FUNCTION_BLOCK FB_InterlockManager

VAR
	aInterlocks: ARRAY[1..50] OF ST_Interlock;
	nIterator: INT := 1;
END_VAR

METHOD execute : BOOL
VAR_INPUT
END_VAR

VAR
	iterator: INT;

	
	Active:			BOOL;
	Bridge:			BOOL;
	SubjectDevice:	POINTER TO FB_BaseDevice;
	SubjectState:	E_DeviceState;
	Signal:			BOOL;
	Description: 	STRING(255);
	HoldSeq:		BOOL;
	InterlockType:	E_InterlockType;
	
	
	
END_VAR

FOR iterator:=1 TO nIterator BY 1 DO
	
	// Update local variable on each loop iteration
	
	Active := aInterlocks[iterator].Active;
	Bridge := aInterlocks[iterator].Bridge;
	SubjectDevice := aInterlocks[iterator].SubjectDevice;
	SubjectState  := aInterlocks[iterator].SubjectState;
	Signal := aInterlocks[iterator].Signal;
	HoldSeq := aInterlocks[iterator].HoldSeq;
	InterlockType := aInterlocks[iterator].InterlockType;
	
	
	IF Signal = TRUE THEN
		
		// Interlock causes the sequence to go into hold (by disabling device)
		// Sequence hold requires operator acknowledgement to resume
		IF  SubjectDevice^.isEnabled() AND HoldSeq AND Bridge <> TRUE THEN
			
			SubjectDevice^.setCommand(StateTarget := SubjectState);
			SubjectDevice^.disable();
			aInterlocks[iterator].Active := TRUE;
		
			
		// Interlock causes device to change state only
		// No operator acknowledgement required 
		ELSIF  SubjectDevice^.isEnabled() AND HoldSeq =FALSE AND Bridge <> TRUE THEN
			
			SubjectDevice^.setCommand(StateTarget := SubjectState);
			aInterlocks[iterator].Active := TRUE;
			
		ELSE
			aInterlocks[iterator].Active := FALSE;
		END_IF
		
	ELSE
		aInterlocks[iterator].Active := FALSE;
	END_IF
END_FOR
END_METHOD

METHOD init : BOOL
VAR_INPUT
END_VAR
// Reset the iterator on each cycle of the machine
nIterator := 1;
END_METHOD

METHOD update : BOOL
VAR_INPUT
	Description:	STRING;
	InterlockType: 	E_InterlockType;
	Subject_Device: POINTER TO FB_BaseDevice;
	Subject_State:	E_DeviceState;
	Signal: 		BOOL;
	HoldSequence: 	BOOL;
END_VAR
aInterlocks[nIterator].HoldSeq := HoldSequence;
aInterlocks[nIterator].InterlockType := InterlockType;
aInterlocks[nIterator].Signal := Signal;
aInterlocks[nIterator].Description := Description;
aInterlocks[nIterator].SubjectDevice := Subject_Device;
aInterlocks[nIterator].SubjectVarID := Subject_Device^.getVarID();
aInterlocks[nIterator].SubjectState := Subject_State;

nIterator := nIterator + 1;
END_METHOD

END_FUNCTION_BLOCK

(* stored: Version 1.1.0.1, ProductVersion 3.1.4024.12
   POU FB_InterlockManager: Id {35055f59-c3c2-4ffb-ab07-3737f8dd7c90}, SpecialFunc None
   Method execute: Id {229a8784-5db6-49d7-805c-74440ccef9e2}
   Method init: Id {9dea35ec-0113-4e40-b16f-f7a26be06aa2}
   Method update: Id {85cfdc67-9c27-4e30-8986-d02f1c1b0c01} *)
